// TwinCAT 3 PLC project Analog_Current_Output
// ProgramVersion: 3.1.4023.0
// libraries:
//   Tc2_Standard, * (Beckhoff Automation GmbH)
//   Tc2_System, * (Beckhoff Automation GmbH)
//   Tc3_Module, * (Beckhoff Automation GmbH)
// project tree:
//   GVLs/ GVL.TcGVL
//   / PlcTask.TcTTO
//   POUs/ MAIN.TcPOU, WriteAnalogOutputCurrent.TcPOU
// real-time tasks:
//   TASK PlcTask: cycle T#10ms, priority 20, ADS port 350
// I/O:
//   DEVICE Dispositivo 1 (EtherCAT), AmsNetId 5.71.198.244.2.1
//     Terminale 1 (EK1200) [EK1200-5000 EtherCAT Power supply (2A E-Bus)]
//       Terminale 2 (EL1008) [EL1008 8Ch. Dig. Input 24V, 3ms]
//       Terminale 3 (EL2008) [EL2008 8Ch. Dig. Output 24V, 0.5A]
//       Terminale 4 (EL3064) [EL3064 4Ch. Ana. Input 0-10V]
//       Terminale 5 (EL4002) [EL4002 2Ch. Ana. Output 0-10V, 12bit]
//       Terminale 6 (EL7031) [EL7031 1Ch. Stepper motor output stage (24V, 1.5A)]
//       Terminale 7 (EL3202) [EL3202 2Ch. Ana. Input PT100 (RTD)]
//       Terminale 8 (EL4022) [EL4022 2Ch. Ana. Output 4-20mA, 12bit]
//       Terminale 9 (EL9011) [EL9011 End Terminal]

CONFIGURATION Analog_Current_Output
    RESOURCE PLC ON TwinCAT3
        TASK PlcTask(INTERVAL := T#10ms, PRIORITY := 20);
        PROGRAM MAIN WITH PlcTask : MAIN;
    END_RESOURCE
END_CONFIGURATION

// ---- GVLs/GVL.TcGVL
{attribute 'qualified_only'}
VAR_GLOBAL
	Analog_Outputs_Curr AT %Q* : ARRAY[1..2] OF INT;
	Analog_Outputs_Curr_Values : ARRAY[1..2] OF REAL;
END_VAR

// ---- POUs/MAIN.TcPOU
PROGRAM MAIN
VAR
	rWriteAnalog1 : REAL;
	rWriteAnalog2 : REAL;
END_VAR

GVL.Analog_Outputs_Curr[1] := REAL_TO_INT((rWriteAnalog1-4)/16*32767);
GVL.Analog_Outputs_Curr[2] := REAL_TO_INT((rWriteAnalog2-4)/16*32767);

END_PROGRAM

// ---- POUs/WriteAnalogOutputCurrent.TcPOU
PROGRAM WriteAnalogOutputCurrent
VAR
	temp: REAL;
END_VAR

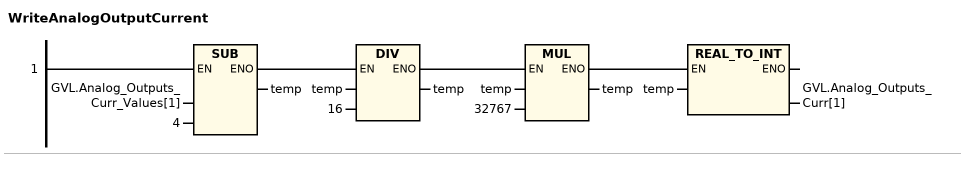
// NETWORK 1
temp := GVL.Analog_Outputs_Curr_Values[1] - 4;
temp := temp / 16;
temp := temp * 32767;
GVL.Analog_Outputs_Curr[1] := REAL_TO_INT(temp);

END_PROGRAM
